// TwinCAT 3 PLC project Punzonatrice_MSF_Efficace
// ProgramVersion: 3.1.4024.0
// libraries:
//   Tc2_Standard, * (Beckhoff Automation GmbH)
//   Tc2_System, * (Beckhoff Automation GmbH)
//   Tc3_Module, * (Beckhoff Automation GmbH)
//   Util, * (System)
// project tree:
//   / PlcTask.TcTTO
//   POUs/HMI/Structs/ ST_HMI.TcDUT
//   POUs/ MAIN.TcPOU
//   POUs/StateMachine/Enums/ E_Step.TcTLEO
//   POUs/StateMachine/FB/ FB_Diagnostic.TcPOU, FB_FSM.TcPOU, FB_ReadCmd.TcPOU, FB_ReadInputs.TcPOU, FB_WriteOutputs.TcPOU, FB_ReadCtrl.TcPOU
//   POUs/StateMachine/ FB_Punzonatrice_Main.TcPOU
//   POUs/StateMachine/Structs/ ST_Cmd.TcDUT, ST_Ctrl.TcDUT, ST_Status.TcDUT, ST_In.TcDUT, ST_out.TcDUT, ST_Params.TcDUT, ST_RawIn.TcDUT, ST_RawOut.TcDUT
// real-time tasks:
//   TASK PlcTask: cycle T#10ms, priority 20, ADS port 350
// motion (NC):
//   TASK NC-Task 1 SAF: cycle T#2ms, priority 4, ADS port 501
//   TASK NC-Task 1 SVB: cycle T#10ms, priority 8, ADS port 511
//   AXIS Asse 1 (id 1)
//     OtherSettings: AllowMotionCmdToSlave=true
//     encoder EncType=4
//       EncPara: MaxCount=#x0000ffff
//         Inc: RefSoftSyncMask=#x0000ffff
//     drive DrvType=24
//       Analog: TorqueSetpointScale=10, ScaleFactorActTorque=0.1
//       TimeComp: TaskDelayCycles=1
//     controller CtrType=1
//       CtrPara: PriorControlFactor=1
//         Observer: BandWidth=20
//   AXIS Asse 2 (id 2)
//     OtherSettings: AllowMotionCmdToSlave=true
//     encoder EncType=4
//       EncPara: MaxCount=#x0000ffff
//         Inc: RefSoftSyncMask=#x0000ffff
//     drive DrvType=24
//       Analog: TorqueSetpointScale=10, ScaleFactorActTorque=0.1
//       TimeComp: TaskDelayCycles=1
//     controller CtrType=1
//       CtrPara: PriorControlFactor=1
//         Observer: BandWidth=20
//   AXIS Asse 3 (id 3)
//     OtherSettings: AllowMotionCmdToSlave=true
//     encoder EncType=4
//       EncPara: MaxCount=#x0000ffff
//         Inc: RefSoftSyncMask=#x0000ffff
//     drive DrvType=24
//       Analog: TorqueSetpointScale=10, ScaleFactorActTorque=0.1
//       TimeComp: TaskDelayCycles=1
//     controller CtrType=1
//       CtrPara: PriorControlFactor=1
//         Observer: BandWidth=20
// I/O:
//   DEVICE Dispositivo 1 (EtherCAT) (disabled), AmsNetId 192.168.56.1.2.1
//     Terminale 1 (EK1200) [EK1200-5000 EtherCAT Power supply (2A E-Bus)]
//       Terminale 2 (EL1809) [EL1809 16Ch. Dig. Input 24V, 3ms]
//       Terminale 3 (EL2809) [EL2809 16Ch. Dig. Output 24V, 0.5A]
//       Terminale 4 (EL3201) [EL3201 1Ch. Ana. Input PT100 (RTD)]
//       Terminale 5 (EL3311) [EL3311 1Ch. Ana. Input Thermocouple (TC)]
//       Terminale 6 (EL3004) [EL3004 4Ch. Ana. Input +/-10V]
//       Terminale 7 (EL1918) [EL1918, 8Ch. Safety Input 24V, TwinSAFE]
//         modules: Module 1 (FSOE), Module 2 (FSLOGIC)
//       Terminale 8 (EL2904) [EL2904, 4 Ch. Safety Output 24V, 0.5A, TwinSAFE]
//         modules: Module 1 (FSOES), Module 2 (DO)
//       Terminale 9 (EL9011) [EL9011 End Terminal]
//   DEVICE Dispositivo 4 (EtherCAT) (disabled), AmsNetId 192.168.56.1.5.1
//     Terminale 10 (EK1100) [EK1100 EtherCAT Coupler (2A E-Bus)]
//       Terminale 11 (EL1809) [EL1809 16Ch. Dig. Input 24V, 3ms]
//       Terminale 12 (EL2809) [EL2809 16Ch. Dig. Output 24V, 0.5A]
//       Terminale 13 (EL1809) [EL1809 16Ch. Dig. Input 24V, 3ms]
//       Terminale 14 (EL2809-0015) [EL2809-0015 16Ch. Dig. Output 24V DC, 0.35A, not short-circuit proof]
//       Terminale 15 (EL7031) [EL7031 1Ch. Stepper motor output stage (24V, 1.5A)]
//       Terminale 7 (EL9011) [EL9011 End Terminal]
// variable links:
//   (this object) <-> Device 4 (EtherCAT)/Term 10 (EK1100)/Term 15 (EL7031)
//     Drive/Inputs/In/nState1 @bit 3 <-> STM Status/Status/Error
//     Drive/Inputs/In/nState1 @bit 5 <-> STM Status/Status/Moving negative
//     Drive/Inputs/In/nState1 @bit 4 <-> STM Status/Status/Moving positive
//     Drive/Inputs/In/nState1 @bit 1 <-> STM Status/Status/Ready
//     Drive/Inputs/In/nState1 <-> STM Status/Status/Ready to enable
//     Drive/Inputs/In/nState1 @bit 6 <-> STM Status/Status/Torque reduced
//     Drive/Inputs/In/nState1 @bit 2 <-> STM Status/Status/Warning
//     Drive/Inputs/In/nState2 @bit 3 <-> STM Status/Status/Digital input 1
//     Drive/Inputs/In/nState2 @bit 4 <-> STM Status/Status/Digital input 2
//     Drive/Inputs/In/nState2 @bit 5 <-> STM Status/Status/Sync error
//     Drive/Inputs/In/nState2 @bit 7 <-> STM Status/Status/TxPDO Toggle
//     Drive/Inputs/In/nState4 @bit 1 <-> WcState/InputToggle
//     Drive/Inputs/In/nState4 <-> WcState/WcState
//     Drive/Outputs/Out/nCtrl1 <-> STM Control/Control/Enable
//     Drive/Outputs/Out/nCtrl1 @bit 2 <-> STM Control/Control/Reduce torque
//     Drive/Outputs/Out/nCtrl1 @bit 1 <-> STM Control/Control/Reset
//     Drive/Outputs/Out/nDataOut2[0] <-> STM Velocity/Velocity
//     Enc/Inputs/In/nDataIn1[0] <-> ENC Status compact/Counter value
//     Enc/Inputs/In/nDataIn2[0] <-> ENC Status compact/Latch value
//     Enc/Inputs/In/nState1 @bit 4 <-> ENC Status compact/Status/Counter overflow
//     Enc/Inputs/In/nState1 @bit 3 <-> ENC Status compact/Status/Counter underflow
//     Enc/Inputs/In/nState1 @bit 1 <-> ENC Status compact/Status/Latch extern valid
//     Enc/Inputs/In/nState1 @bit 2 <-> ENC Status compact/Status/Set counter done
//     Enc/Inputs/In/nState2 @bit 4 <-> ENC Status compact/Status/Status of extern latch
//     Enc/Inputs/In/nState2 @bit 5 <-> ENC Status compact/Status/Sync error
//     Enc/Inputs/In/nState2 @bit 7 <-> ENC Status compact/Status/TxPDO Toggle
//     Enc/Inputs/In/nState4 @bit 1 <-> WcState/InputToggle
//     Enc/Inputs/In/nState4 <-> WcState/WcState
//     Enc/Outputs/Out/nCtrl1 @bit 3 <-> ENC Control compact/Control/Enable latch extern on negative edge
//     Enc/Outputs/Out/nCtrl1 @bit 1 <-> ENC Control compact/Control/Enable latch extern on positive edge
//     Enc/Outputs/Out/nCtrl1 @bit 2 <-> ENC Control compact/Control/Set counter
//     Enc/Outputs/Out/nDataOut1[0] <-> ENC Control compact/Set counter value
//   Punzonatrice_MSF_Efficace Instance <-> Device 1 (EtherCAT)/Term 1 (EK1200)/Term 2 (EL1809)
//     PlcTask Inputs/MAIN.stRawIn.bAck <-> Channel 7/Input
//     PlcTask Inputs/MAIN.stRawIn.bEmg <-> Channel 8/Input
//     PlcTask Inputs/MAIN.stRawIn.bFc{1..4} <-> Channel {1..4}/Input  (4 links)
//     PlcTask Inputs/MAIN.stRawIn.bStart <-> Channel 5/Input
//     PlcTask Inputs/MAIN.stRawIn.bStop <-> Channel 6/Input
//   Punzonatrice_MSF_Efficace Instance <-> Device 1 (EtherCAT)/Term 1 (EK1200)/Term 3 (EL2809)
//     PlcTask Outputs/MAIN.stRawOut.bLAck <-> Channel 7/Output
//     PlcTask Outputs/MAIN.stRawOut.bLStart <-> Channel 5/Output
//     PlcTask Outputs/MAIN.stRawOut.bLStop <-> Channel 6/Output
//     PlcTask Outputs/MAIN.stRawOut.bQ{1..4} <-> Channel {1..4}/Output  (4 links)

CONFIGURATION Punzonatrice_MSF_Efficace
    RESOURCE PLC ON TwinCAT3
        TASK PlcTask(INTERVAL := T#10ms, PRIORITY := 20);
        PROGRAM MAIN WITH PlcTask : MAIN;
    END_RESOURCE
END_CONFIGURATION

// ---- POUs/HMI/Structs/ST_HMI.TcDUT
TYPE ST_HMI :
STRUCT
	bStart	:	BOOL;  // N.O.
	bStop	:	BOOL;  // N.O.
END_STRUCT
END_TYPE

// ---- POUs/StateMachine/Enums/E_Step.TcTLEO
{attribute 'qualified_only'}
{attribute 'strict'}
{attribute 'to_string'}
TYPE E_Step :
(
	// Special steps
	NoStep := -32767,	// No step
	Unknown := -32000,	// Unknown step
	
	// Not Enabled or Errors
	NeOrError := -990,	// Not enabled or at fault //
	
	// Recovery
	Recovering := 990,	// Restore After Failure //

	// Stopping
	Stopping := 900,	// Nominal shutdown //
	
	// Stop
	Stop := 0, 			// S0 Stop //
	
	// Working steps
	RecoverPunch := 50,		// S1 Lift the punch at restart //
	WaitObject := 100,		// S2 Waiting for object //
	DelayToFeeding := 120,	// S3 delay before feeding  //
	Loading := 200,			// S4 Object Transfer //
	LowerPunch := 300,		// S5 Lower the punch //
	LiftPunch := 400,		// S6 Lift the punch //
	Unloading := 500,		// S7 Outgoing object discharge //
	DelayOnUnloading := 520	// S8 delay after unloading //
   
);
END_TYPE
//  NoStep = '-32767'
//  Unknown = '-32000'
//  NeOrError = '-990'

// ---- POUs/StateMachine/Structs/ST_Cmd.TcDUT
TYPE ST_Cmd :
STRUCT
	bAck	:	BOOL;	// Alarm Recognition
	bStop	:	BOOL;	// Stop the machine
	bStart	:	BOOL;	// Starts the machine	
END_STRUCT
END_TYPE

// ---- POUs/StateMachine/Structs/ST_Ctrl.TcDUT
TYPE ST_Ctrl :
STRUCT
	bEmergency	:	BOOL;	// Emergency. It must be TRUE for the machine to operate
	bEnable		:	BOOL;	// Machine enablement. It must be TRUE for the machine to operate	
END_STRUCT
END_TYPE

// ---- POUs/StateMachine/Structs/ST_Status.TcDUT
TYPE ST_Status :
STRUCT
	bCritical : BOOL;			// The machine has at least one active critical condition
	bError : BOOL;				// The machine has at least one active error condition	
	bWarning : BOOL;			// The machine has at least one active signal	
	bInfo : BOOL;				// The machine has at least one active piece of information			
	bVerbose : BOOL;			// The machine has at least one active message
	bFailure : BOOL;			// The machine has broken down (critical + error)	

	eStep : E_Step;				// Finite State Machine step
	strStep : STRING;			// step described as text
	tStepTime : TIME;			// elapsed time on each state machine step/state
	eErrorStep : E_Step;		// Step in which the error was generated
	nErrorID : DINT;			// Error code	
END_STRUCT
END_TYPE

// ---- POUs/StateMachine/Structs/ST_In.TcDUT
TYPE ST_In :
STRUCT
	// Digital Inputs
	bStart	:	BOOL;	// start button active HIGH
	bStop	:	BOOL;	// stop button active HIGH
	bEmg	:	BOOL;	// emergency button active LOW
	bAck	:	BOOL;	// error acknowledge button active HIGH
	bFc1	:	BOOL;	// proximity sensor on conveyor input active HIGH
	bFc2	:	BOOL;	// proximity sensor on conveyor workplace active HIGH
	bFc3	:	BOOL;	// proximity sensor at punch top active HIGH
	bFc4	:	BOOL;	// proximity sensor at punch bottom active HIGH
END_STRUCT
END_TYPE

// ---- POUs/StateMachine/Structs/ST_out.TcDUT
TYPE ST_out :
STRUCT
	// Digital Outputs
	bFixedGreen		:	BOOL;	// machine running light green indicator
	bBlinkingGreen	:	BOOL;	// machine stopping blinking light green indicator	
	bFixedRed		:	BOOL;	// machine stopped light red indicator
	bBlinkingRed	:	BOOL;	// blinking red indicator
	bFixedOrange	:	BOOL;	// recovery light orange indicator	
	bBlinkingOrange	:	BOOL;	// blinking orange indicator
	bQ1				:	BOOL;	// loading conveyor motor
	bQ2				:	BOOL;	// unloading conveyor motor
	bQ3				:	BOOL;	// lower the punch piston
	bQ4				:	BOOL;	// lift the punch piston
END_STRUCT
END_TYPE

// ---- POUs/StateMachine/Structs/ST_Params.TcDUT
TYPE ST_Params :
STRUCT
	// machine parameters
	tLoadingDelay	:	TIME := T#3S;
	tUnloadingDelay	:	TIME := T#3S;
	tMaxTravelTime	: TIME := T#5S;  // max travel time on conveyor
	tMaxPunchMoveTime : TIME := T#3S; // max punch moving time
	tStoppingDelay	:	TIME := T#2s;
END_STRUCT
END_TYPE

// ---- POUs/StateMachine/Structs/ST_RawIn.TcDUT
TYPE ST_RawIn :
STRUCT
	// Physical digital Inputs
	bStart	AT %I*	:	BOOL;	// start button (N.O. contact)
	bStop	AT %I*	:	BOOL;	// stop button (N.C. contact)
	bEmg	AT %I*	:	BOOL;	// emergency button (N.C. contact)
	bAck	AT %I*	:	BOOL;	// error acknowledge button (N.O. contact)
	bFc1	AT %I*	:	BOOL;	// proximity sensor on conveyor input (N.C. contact)
	bFc2	AT %I*	:	BOOL;	// proximity sensor on conveyor workplace (N.C. contact)
	bFc3	AT %I*	:	BOOL;	// proximity sensor at punch top (N.O. contact)
	bFc4	AT %I*	:	BOOL;	// proximity sensor at punch bottom (N.O. contact)	
END_STRUCT
END_TYPE

// ---- POUs/StateMachine/Structs/ST_RawOut.TcDUT
TYPE ST_RawOut :
STRUCT
	// Physical digital Outputs
	bLStart	AT %Q*	:	BOOL;	// machine running light green indicator
	bLStop	AT %Q*	:	BOOL;	// machine stopped light red indicator
	bLAck	AT %Q*	:	BOOL;	// recovery light orange indicator	
	bQ1		AT %Q*	:	BOOL;	// loading conveyor motor
	bQ2		AT %Q*	:	BOOL;	// unloading conveyor motor
	bQ3		AT %Q*	:	BOOL;	// lower the punch piston
	bQ4		AT %Q*	:	BOOL;	// lift the punch piston	
END_STRUCT
END_TYPE

// ---- POUs/MAIN.TcPOU
PROGRAM MAIN
VAR
	bInitialized : BOOL;
	
	fbGetCurTaskIndex : GETCURTASKINDEX;		
	tTaskCycleTime : UDINT;					// tempo di ciclo della task in microsecondi
	tTaskExecTime : UDINT;					// tempo di esecuzione della task in microsecondi
	tTaskMaxExecTime : UDINT;				// tempo massimo di esecuzione della task in microsecondi

// machine I/Os 	
// inputs
	stIn		:	ST_In;
	stRawIn		:	ST_RawIn;
	stHmi		:	ST_HMI;

// outputs
	stOut		:	ST_Out;
	stRawOut	:	ST_RawOut;	
	
// state machine internals, useful for debugging
	stStatus	: 	ST_Status;
	
// machine controls
	stCtrl		:	ST_Ctrl;

// full machine
  fbPunzonatrice	:	FB_Punzonatrice_Main();
  
END_VAR

IF NOT bInitialized THEN
	// Get the Cycle Time of the task to which this PRG is assigned (it will then be shared with the State Machine)
	fbGetCurTaskIndex();
	tTaskCycleTime := _TaskInfo[fbGetCurTaskIndex.index].CycleTime / 10;	// CycleTime is expressed in multiples of 100ns
	bInitialized := TRUE;
	
ELSE
	(* task time *)
	tTaskExecTime := _TaskInfo[fbGetCurTaskIndex.index].LastExecTime / 10;		// ExecTime is expressed in multiples of 100ns
	IF tTaskExecTime > tTaskMaxExecTime THEN
			tTaskMaxExecTime := tTaskExecTime;
	END_IF;	
	
	(* machine *)
	fbPunzonatrice(
		bEnable:= TRUE, 
		tTaskCycleTime:= tTaskExecTime, 
		nId:= 0, 
		bHwError:= FALSE, 
		stRawIn:= stRawIn, 
		stIn:= stIn, 
		stRawOut:= stRawOut, 
		stOut:= stOut, 
		stCtrl:= stCtrl, 
		stHmi := stHmi,
		stStatus:= stStatus);
	
END_IF

END_PROGRAM

// ---- POUs/StateMachine/FB_Punzonatrice_Main.TcPOU
FUNCTION_BLOCK FB_Punzonatrice_Main
VAR_INPUT
	(* main inputs to the state machine *)
	bEnable			: BOOL;		// state machine enable
	tTaskCycleTime	: UDINT;
	nId				: USINT;	
	bHwError		: BOOL;		
END_VAR
VAR_OUTPUT
END_VAR
VAR_IN_OUT
	(* machine I/Os *)
	stRawIn		:	ST_RawIn;
	stIn		:	ST_In;
	stRawOut	:	ST_RawOut;
	stOut		:	ST_Out;
	stCtrl		:	ST_Ctrl;
	
	(* HMI inputs *)
	stHmi		:	ST_HMI;
	
	(* state machine internals, useful for debugging  *)
	stStatus	:	ST_Status;	
END_VAR
VAR
	bInitialized	: 	BOOL;		// FB initialization
	stCmd			:	st_Cmd;
	stParams		:	ST_Params;	
	errno			:	INT;
	fbReadCmd		:	FB_ReadCmd;
	fbReadCtrl		:	FB_ReadCtrl;
	fbReadIn		:	FB_ReadInputs;
	fbDiagnostic	:	FB_Diagnostic;
	fbStateMachine	:	FB_FSM;
	fbWriteOut		:	FB_WriteOutputs;
END_VAR

IF NOT bInitialized THEN
	// start-up operations
	bInitialized := TRUE;
ELSE
	// 01. Read inputs, controls, parameters and commands
	fbReadIn( stRawIn := stRawIn,
			  stIn => stIn);
			 
	fbReadCtrl( nId:= nId,
				bEnable:= bEnable,
				stIn:= stIn,
				stCtrl=> stCtrl);
				
	fbReadCmd( stIn:= stIn, 
			   stHmi := stHmi,
			   stCmd=> stCmd);
			   
	// 02. events management fbDiagnostic
	fbDiagnostic(
	stIn:= stIn, 
	stOut:= stOut, 
	stParams:= stParams, 
	stCtrl:= stCtrl, 
	bHwError:= bHwError, 
	bAck:= stCmd.bAck, 
	stStatus:= stStatus);
	
	stStatus.bCritical := fbDiagnostic.bCritical;
	stStatus.bError := fbDiagnostic.bError;
	stStatus.bWarning := fbDiagnostic.bWarning;
	stStatus.bInfo := fbDiagnostic.bInfo;
	stStatus.bVerbose := fbDiagnostic.bVerbose;
	stStatus.bFailure := fbDiagnostic.bFailure;
	stOut.bBlinkingRed := fbDiagnostic.bCritical;
	stOut.bBlinkingOrange := fbDiagnostic.bBlinking;
	stOut.bFixedOrange := fbDiagnostic.bFixed;
	
	// 03. main finite state machine
	fbStateMachine(
		stIn:= stIn, 
		stCtrl:= stCtrl, 
		stCmd:= stCmd, 
		stParams:= stParams, 
		stStatus:= stStatus
	);
	stStatus.eStep := fbStateMachine.eStep;
	stStatus.strStep := TO_STRING(stStatus.eStep);
	stStatus.tStepTime := fbStateMachine.tStepTime;
	stStatus.eErrorStep := fbStateMachine.eErRstep; 
	stStatus.nErrorID := fbStateMachine.nErrId;
	
	stOut.bFixedGreen := fbStateMachine.bFixedGreen;
	stOut.bBlinkingGreen := fbStateMachine.bBlinkingGreen;
	stOut.bFixedRed := fbStateMachine.bFixedRed;
	stOut.bBlinkingRed := fbStateMachine.bBlinkingRed;
	stOut.bFixedOrange := fbStateMachine.bFixedOrange;
	stOut.bBlinkingOrange := fbStateMachine.bBlinkingOrange;
	
	stOut.bQ1 := fbStateMachine.bQ1;
	stOut.bQ2 := fbStateMachine.bQ2;
	stOut.bQ3 := fbStateMachine.bQ3;
	stOut.bQ4 := fbStateMachine.bQ4;	

    // 04. secondary state machines
	
	// 05. write outputs and machine information
	fbWriteOut( stOut:= stOut, 
				stRawOut:= stRawOut);
				
	// 06. end - other operations
	
				
END_IF

END_FUNCTION_BLOCK

// ---- POUs/StateMachine/FB/FB_ReadCmd.TcPOU
FUNCTION_BLOCK FB_ReadCmd
VAR_INPUT
	stIn	:	ST_In;
	stHmi	:	ST_HMI;
END_VAR
VAR_OUTPUT
	stCmd	:	ST_Cmd;
END_VAR
VAR
//	fbRtStart	: R_TRIG;
//	fbRtStop	: R_TRIG;
	fbTpStart	: TP;
	fbTpStop	: TP;	
	fbTpAck		: TP;	
END_VAR

// filters on input button
fbTpStart( IN := stIn.bStart, PT := T#50MS );
fbTpStop( IN := stIn.bStop, PT := T#50MS );
fbTpAck( IN := stIn.bAck, PT := T#50MS );

//stCmd.bStart	:= fbRtStart.Q;
//stCmd.bStop		:= fbRtStop.Q;
stCmd.bStart	:= fbTpStart.Q OR stHmi.bStart;
stCmd.bStop		:= fbTpStop.Q OR stHmi.bStop;
stCmd.bAck		:= fbTpAck.Q;

END_FUNCTION_BLOCK

// ---- POUs/StateMachine/FB/FB_ReadCtrl.TcPOU
FUNCTION_BLOCK FB_ReadCtrl
VAR_INPUT
	nId:	INT;
	bEnable : BOOL;
	stIn : ST_In;
END_VAR
VAR_OUTPUT
	stCtrl : ST_Ctrl;
END_VAR
VAR
	fbTonStartup: TON;
END_VAR

fbTonStartup(IN := TRUE, PT := T#3S);
stCtrl.bEmergency := stIn.bEmg;
stCtrl.bEnable := fbTonStartup.Q AND bEnable;

END_FUNCTION_BLOCK

// ---- POUs/StateMachine/FB/FB_ReadInputs.TcPOU
FUNCTION_BLOCK FB_ReadInputs
VAR_INPUT
END_VAR
VAR_IN_OUT
	stRawIn		:	ST_RawIn;
END_VAR
VAR_OUTPUT
	stIn		:	ST_In;
END_VAR
VAR
END_VAR

// digital
stIn.bEmg := stRawIn.bEmg;   // NOTA: Emg è sempre attivo basso
stIn.bStart := stRawIn.bStart;
stIn.bStop := NOT stRawIn.bStop;
stIn.bAck := stRawIn.bAck;
stIn.bFc1 := NOT stRawIn.bFc1;
stIn.bFc2 := NOT stRawIn.bFc2;
stIn.bFc3 := stRawIn.bFc3;
stIn.bFc4 := stRawIn.bFc4;

END_FUNCTION_BLOCK

// ---- POUs/StateMachine/FB/FB_Diagnostic.TcPOU
FUNCTION_BLOCK FB_Diagnostic
VAR_INPUT
	stIn : ST_In;
	stOut : ST_Out;
	stParams : ST_Params;
	stCtrl : ST_Ctrl;
	bHwError : BOOL;
	bAck : BOOL;
	stStatus : ST_Status;	
END_VAR
VAR_IN_OUT
END_VAR
VAR_OUTPUT
	bCritical	: BOOL;
	bError		: BOOL;
	bWarning	: BOOL;
	bInfo		: BOOL;
	bVerbose	: BOOL;
	bFailure	: BOOL;
	bBlinking	: BOOL;
	bFixed		: BOOL;
END_VAR
VAR
END_VAR

// on Ack, reset holding conditions
IF bAck THEN
	bCritical := FALSE;
	bError := FALSE;
	bWarning := FALSE;
	bInfo := FALSE;
	bVerbose := FALSE;
	bBlinking := FALSE;
END_IF

// update holding conditions
bFailure := bCritical OR bError;

bBlinking := bFailure;
bFixed := bWarning;

END_FUNCTION_BLOCK

// ---- POUs/StateMachine/FB/FB_FSM.TcPOU
FUNCTION_BLOCK FB_FSM
VAR_INPUT
	stIn		:	ST_In;
	stCtrl		:	ST_Ctrl;
	stCmd		:	ST_Cmd;
	stParams	:	ST_Params;
	stStatus	:	ST_Status;
END_VAR

VAR_OUTPUT
	eStep		:	E_Step;
	tStepTime	:	TIME;
	eErrStep	:	E_Step;
	nErrId		:	DINT;
	
	// Digital Outputs
	bFixedGreen		:	BOOL;	// machine running light green indicator
	bBlinkingGreen	:	BOOL;	// machine stopping blinking green indicator
	bFixedRed		:	BOOL;	// machine stopped light red indicator
	bBlinkingRed	:	BOOL;	// blinking red indicator
	bFixedOrange	:	BOOL;	// recovery light orange indicator	
	bBlinkingOrange	:	BOOL;	// blinking orange indicator
	bQ1				:	BOOL;	// loading conveyor motor
	bQ2				:	BOOL;	// unloading conveyor motor
	bQ3				:	BOOL;	// lower the punch piston
	bQ4				:	BOOL;	// lift the punch piston	
END_VAR

VAR_IN_OUT

END_VAR

VAR
	bInitialized :  BOOL;
	eNewstep :  E_Step;
	bEntryact :  BOOL;
	fbTonStep :  TON;
	
	(* filters on other input from plant *)
	fbTonPacketIn : TON();		// Filter on the input object presence signal
	fbRtPacketIn : R_TRIG();	// Presence of Incoming Object (rise edge)
	fbTonPacketOut : TON();		// Filter on the object discharge signal
	fbRtPacketOut: R_TRIG();	// Object Discharge (rise edge)
	
	(* filters on stop input *)
	//fbFtStop : F_TRIG;		// Stop control (fall edge)
	bStopRequest : BOOL;		// Stop request
	
	// object on conveyor
	bConveyorLoaded	:	BOOL;


END_VAR

IF NOT bInitialized THEN
	(* here you can wait events from other controllers *)
	eNewStep := E_Step.NoStep;
	eStep := E_Step.Stop;
	bEntryact := FALSE;
	bInitialized := TRUE;
ELSE
	// --- FSM Cyclical Code ----------------------------------------------
	
	// update of the enabling conditions (bStop, alarms, etc.)
    //enable := stCtrl.bEnable AND bStop AND bEmg;
	
	// 1. FSM Preamble ----------------------------------------------------

    // 1.a State machine disabled or failure
	IF NOT stCtrl.bEnable OR NOT stCtrl.bEmergency OR stStatus.bFailure THEN
		eNewStep := E_Step.NeOrError;
	END_IF

	// 1.b Update eStep with the required step to perform
	//     and set bEntryact to FALSE in order to enable the Entry action
	IF eNewstep <> E_Step.NoStep THEN
		eStep := eNewstep;
		eNewstep := E_Step.NoStep;
		bEntryact := FALSE;
	END_IF;

	// 1.c Do filters on signals	
	fbTonPacketIn(IN := stIn.bFc1, PT := T#100MS);	// Object Presence Sensor Filter on Loading Platform
	fbTonPacketOut(IN := stIn.bFc2, PT := T#100MS);	// Object Presence Sensor Filter on Unloading Platform	
	
	//     Do edge detection
	fbRtPacketIn(CLK := fbTonPacketIn.Q);		// Edge detection on Loading Platform
	fbRtPacketOut(CLK := fbTonPacketOut.Q);		// Edge detection on Unloading Platform	
	
	//fbFtStop(CLK := bStop);						// Active edge of the Stop control
	
	// Do requests, for example to stop the machine
	IF stCmd.bStop THEN
		bStopRequest := TRUE;
	END_IF
	
	
	// 2. The main switch-case ---------------------------------------------------
	CASE eStep OF
		// not Enabled or Error -----------------------
		E_Step.NeOrError :
			// on entry action
			IF NOT bEntryact THEN
				stStatus.bFailure := TRUE;
				bEntryact := TRUE;
			END_IF
			
			// body
			bFixedGreen := TRUE;
			bFixedRed := FALSE;
			bBlinkingRed := TRUE;
			bFixedOrange := FALSE;
			bBlinkingOrange := FALSE;
			
			bQ1 := FALSE;
			bQ2 := FALSE;
			bQ3 := FALSE;
			bQ4 := FALSE;			
			
			// next state transition
			IF stCtrl.bEnable THEN
				IF stCmd.bAck THEN
					eNewStep := E_Step.Recovering;
				END_IF
			END_IF
		
			// on exit action
			IF eNewStep <> E_Step.NoStep THEN
				nErrId := 0;
				eErrStep := E_Step.NoStep;
			END_IF
			
		// Recovering ---------------------------------			
		E_Step.Recovering :
			// on entry action
			IF NOT bEntryact THEN
				bEntryact := TRUE;
			END_IF
			
			// body
			bFixedGreen := TRUE;
			bFixedRed := FALSE;
			bBlinkingRed := FALSE;
			bFixedOrange := FALSE;
			bBlinkingOrange := TRUE;
			
			bQ1 := FALSE;
			bQ2 := bConveyorLoaded AND (tStepTime > T#500MS);
			bQ3 := NOT(stIn.bFc3);
			bQ4 := FALSE;
			
			// next state transition
			IF stCtrl.bEnable THEN
				IF NOT(stStatus.bFailure) THEN
					IF (bConveyorLoaded AND stIn.bFc1 AND stIn.bFc3) OR ( NOT(bConveyorLoaded) AND stIn.bFc3 ) OR (tStepTime > stParams.tMaxTravelTime) THEN
						eNewStep := E_Step.Stopping;
					END_IF
				END_IF				
			END_IF
			
			// on exit action
			IF eNewStep <> E_Step.NoStep THEN
				stStatus.bFailure := FALSE;
			END_IF			

		// Stopping -----------------------------------
		E_Step.Stopping :
			// on entry action
			IF NOT bEntryact THEN
				bEntryact := TRUE;
			END_IF
			
			// body
			bFixedGreen := FALSE;
			bBlinkingGreen := TRUE;
			bFixedRed := FALSE;
			bBlinkingRed := FALSE;
			bFixedOrange := FALSE;
			bBlinkingOrange := FALSE;
			
			bQ1 := FALSE;
			bQ2 := FALSE;
			bQ3 := FALSE;
			bQ4 := FALSE;
			
			// next state transition
			IF tStepTime >= stParams.tStoppingDelay THEN
				eNewStep := E_Step.Stop;
			END_IF
			
			// on exit action
			IF eNewStep <> E_Step.NoStep THEN
				;
			END_IF
			
		// Stop ---------------------------------------
		E_Step.Stop :
			// on entry action
			IF NOT bEntryact THEN
				bStopRequest := FALSE;
				bConveyorLoaded := FALSE;
				bEntryact := TRUE;
			END_IF
			
			// body
			bFixedGreen := FALSE;
			bBlinkingGreen := FALSE;
			bFixedRed := TRUE;
			bBlinkingRed := FALSE;
			bFixedOrange := FALSE;
			bBlinkingOrange := FALSE;
			
			bQ1 := FALSE;
			bQ2 := FALSE;
			bQ3 := FALSE;
			bQ4 := FALSE;
			
			// next state transition
			IF NOT stCmd.bStop AND stCmd.bStart THEN
				IF NOT(stIn.bFc3) THEN
					eNewStep := E_Step.RecoverPunch;
				ELSE
					eNewStep := E_Step.WaitObject;
				END_IF
			END_IF
			
			// on exit action
			IF eNewStep <> E_Step.NoStep THEN
				;
			END_IF

		// Recover Punch ------------------------------------
		E_Step.RecoverPunch :
			// on entry action
			IF NOT bEntryact THEN
				//bConveyorLoaded := FALSE;
				bEntryact := TRUE;
			END_IF
			
			// body
			bFixedGreen := TRUE;
			bBlinkingGreen := FALSE;
			bFixedRed := FALSE;
			bBlinkingRed := FALSE;
			bFixedOrange := FALSE;
			bBlinkingOrange := TRUE;
			
			bQ1 := FALSE;
			bQ2 := FALSE;
			bQ3 := NOT(stIn.bFc3);
			bQ4 := FALSE;
			
			// next state transition
			IF bStopRequest THEN
				eNewStep := E_Step.Stopping;
			ELSIF stIn.bFc3 THEN
				eNewStep := E_Step.WaitObject;
			END_IF
			
			// on exit action
			IF eNewStep <> E_Step.NoStep THEN
				;
			END_IF			
			
		// Waiting for new object -----------------------------
		E_Step.WaitObject :
			// on entry action
			IF NOT bEntryact THEN
				//bConveyorLoaded := FALSE;
				bEntryact := TRUE;
			END_IF
			
			// body
			bFixedGreen := TRUE;
			bBlinkingGreen := FALSE;
			bFixedRed := FALSE;
			bBlinkingRed := FALSE;
			bFixedOrange := FALSE;
			bBlinkingOrange := FALSE;
			
			bQ1 := FALSE;
			bQ2 := FALSE;
			bQ3 := FALSE;
			bQ4 := FALSE;
			
			// next state transition
			IF bStopRequest THEN
				eNewStep := E_Step.Stopping;
			ELSIF fbRtPacketIn.Q THEN
				eNewStep := E_Step.DelayToFeeding;
			END_IF
			
			// on exit action
			IF eNewStep <> E_Step.NoStep THEN
				;
			END_IF	

		// A little delay before feeding -----------------------
		E_Step.DelayToFeeding :
			// on entry action
			IF NOT bEntryact THEN
				bConveyorLoaded := TRUE;
				bEntryact := TRUE;
			END_IF
			
			// body
			bFixedGreen := TRUE;
			bBlinkingGreen := FALSE;
			bFixedRed := FALSE;
			bBlinkingRed := FALSE;
			bFixedOrange := FALSE;
			bBlinkingOrange := FALSE;
			
			bQ1 := FALSE;
			bQ2 := FALSE;
			bQ3 := FALSE;
			bQ4 := FALSE;
			
			// next state transition
			IF bStopRequest THEN
				eNewStep := E_Step.Stopping;
			ELSIF tStepTime >= stParams.tLoadingDelay THEN
				eNewStep := E_Step.Loading;
			END_IF
			
			// on exit action
			IF eNewStep <> E_Step.NoStep THEN
				;
			END_IF	
			

		// Transfer Object below the punch -----------
		E_Step.Loading :
			// on entry action
			IF NOT bEntryact THEN
				bConveyorLoaded := TRUE;
				bEntryact := TRUE;
			END_IF
			
			// body
			bFixedGreen := TRUE;
			bBlinkingGreen := FALSE;
			bFixedRed := FALSE;
			bBlinkingRed := FALSE;
			bFixedOrange := FALSE;
			bBlinkingOrange := FALSE;
			
			bQ1 := TRUE;
			bQ2 := FALSE;
			bQ3 := FALSE;
			bQ4 := FALSE;
			
			// next state transition
			// e se la macchina non fosse più abilitata?
			IF fbRtPacketOut.Q THEN
				eNewStep := E_Step.LowerPunch;
			ELSIF tStepTime >= stParams.tMaxTravelTime THEN
				eNewStep := E_Step.NeOrError;
			END_IF
			
			// on exit action
			IF eNewStep <> E_Step.NoStep THEN
				;
			END_IF


		// Lower the punch ----------------------
		E_Step.LowerPunch :
			// on entry action
			IF NOT bEntryact THEN
				bConveyorLoaded := TRUE;
				bEntryact := TRUE;
			END_IF
			
			// body
			bFixedGreen := TRUE;
			bBlinkingGreen := FALSE;
			bFixedRed := FALSE;
			bBlinkingRed := FALSE;
			bFixedOrange := FALSE;
			bBlinkingOrange := FALSE;
			
			bQ1 := FALSE;
			bQ2 := FALSE;
			bQ3 := FALSE;
			bQ4 := NOT(stIn.bFc4);
			
			// next state transition
			IF stIn.bFc4 THEN
				eNewStep := E_Step.LiftPunch;
			ELSIF tStepTime >= stParams.tMaxPunchMoveTime THEN
				eNewStep := E_Step.NeOrError;
			END_IF
			
			// on exit action
			IF eNewStep <> E_Step.NoStep THEN
				;
			END_IF


		// Lift the punch ----------------------
		E_Step.LiftPunch :
			// on entry action
			IF NOT bEntryact THEN
				bConveyorLoaded := TRUE;
				bEntryact := TRUE;
			END_IF
			
			// body
			bFixedGreen := TRUE;
			bBlinkingGreen := FALSE;
			bFixedRed := FALSE;
			bBlinkingRed := FALSE;
			bFixedOrange := FALSE;
			bBlinkingOrange := FALSE;
			
			bQ1 := FALSE;
			bQ2 := FALSE;
			bQ3 := NOT(stIn.bFc3);
			bQ4 := FALSE;
			
			// next state transition
			IF stIn.bFc3 THEN
				eNewStep := E_Step.Unloading;
			ELSIF tStepTime >= stParams.tMaxPunchMoveTime THEN
				eNewStep := E_Step.NeOrError;
			END_IF
			
			// on exit action
			IF eNewStep <> E_Step.NoStep THEN
				;
			END_IF

		// Outgoing object discharge ----------------------
		E_Step.Unloading :
			// on entry action
			IF NOT bEntryact THEN
				bConveyorLoaded := TRUE;
				bEntryact := TRUE;
			END_IF
			
			// body
			bFixedGreen := TRUE;
			bBlinkingGreen := FALSE;
			bFixedRed := FALSE;
			bBlinkingRed := FALSE;
			bFixedOrange := FALSE;
			bBlinkingOrange := FALSE;
			
			bQ1 := FALSE;
			bQ2 := TRUE;
			bQ3 := FALSE;
			bQ4 := FALSE;
			
			// next state transition
			IF fbRtPacketIn.Q THEN
				eNewStep := E_Step.DelayOnUnloading;
			ELSIF tStepTime >= stParams.tMaxTravelTime THEN
				eNewStep := E_Step.NeOrError;
			END_IF
			
			// on exit action
			IF eNewStep <> E_Step.NoStep THEN
				;
			END_IF


		// delay after unloading ----------------------
		E_Step.DelayOnUnloading :
			// on entry action
			IF NOT bEntryact THEN
				bConveyorLoaded := TRUE;
				bEntryact := TRUE;
			END_IF
			
			// body
			bFixedGreen := TRUE;
			bBlinkingGreen := FALSE;
			bFixedRed := FALSE;
			bBlinkingRed := FALSE;
			bFixedOrange := FALSE;
			bBlinkingOrange := FALSE;
			
			bQ1 := FALSE;
			bQ2 := FALSE;
			bQ3 := FALSE;
			bQ4 := FALSE;
			
			// next state transition
			IF bStopRequest THEN
				eNewStep := E_Step.Stopping;
			ELSIF tStepTime >= stParams.tUnloadingDelay AND NOT(stIn.bFc1) THEN
				eNewStep := E_Step.WaitObject;
			END_IF
			
			// on exit action
			IF eNewStep <> E_Step.NoStep THEN
				;
			END_IF

		
//--------------------			
		
			
	ELSE
		// this happens also if we forget to code one step 
		eNewstep := E_Step.NeOrError;
		eErrStep := E_Step.Unknown;
		nErrId := -9;
	END_CASE;
	
	// 3. FSM Epilogue ------------------------------------------------------
	// 3.1 Calling Auxiliary FBs
	
	// 3.2 Elapsed time into the current step
	fbTonStep(IN := (eNewstep = E_Step.NoStep), PT := T#500H );
	tStepTime := fbTonStep.ET;
	
END_IF

END_FUNCTION_BLOCK

// ---- POUs/StateMachine/FB/FB_WriteOutputs.TcPOU
FUNCTION_BLOCK FB_WriteOutputs
VAR_INPUT
	stOut		:	ST_Out;
END_VAR
VAR_IN_OUT
	stRawOut	:	ST_RawOut;	
END_VAR
VAR
	fbBlink		:	BLINK;	
END_VAR

// blinking
fbBlink(ENABLE:= TRUE, TIMELOW:= T#500MS, TIMEHIGH:= T#500MS);

// lights on control panel
IF stOut.bBlinkingOrange THEN
	stRawOut.bLAck := fbBlink.OUT;
ELSE
	IF stOut.bFixedOrange THEN
		stRawOut.bLAck := TRUE;
	ELSE
		stRawOut.bLAck := FALSE;		
	END_IF
END_IF

IF stOut.bBlinkingGreen THEN
	stRawOut.bLStart := fbBlink.OUT;
ELSE
	IF stOut.bFixedGreen THEN
		stRawOut.bLStart := TRUE;
	ELSE
		stRawOut.bLStart := FALSE;		
	END_IF
END_IF

IF stOut.bBlinkingRed THEN
	stRawOut.bLStop := fbBlink.OUT;
ELSE
	IF stOut.bFixedRed THEN
		stRawOut.bLStop := TRUE;
	ELSE
		stRawOut.bLStop := FALSE;		
	END_IF
END_IF


// other digital outputs
stRawOut.bQ1 := stOut.bQ1;
stRawOut.bQ2 := stOut.bQ2;
stRawOut.bQ3 := stOut.bQ3;
stRawOut.bQ4 := stOut.bQ4;

END_FUNCTION_BLOCK
